ABB RobotStudio station: smART_ABB_robotstudio_model.rsstn

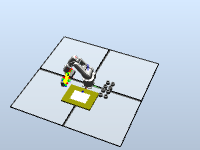
Station smART_v3 (saved by RobotStudio 6.7.7850.130)
Controller IRB120_3kg_0.58m
  mechanical unit ROB_1: IRB120_3_58__01, 6 joints, base frame (0, 0, 0) mm
Layout (positions relative to the parent item):
  - IRB120_3_58__01 [mechanism, from Robots\IRB120_3_58_G_01.rslib] at (0, 0, 0) mm; joint values [-1.4746, 0.7594, 0.252, 0.0074, 0.5575, -0.7708] (rad or m)
  - Grundplatte [part] at (-350, 0, 0) mm
  - Malplatte [part]
  - Papier [part]
  - Waschstation [part]
  - pen [mechanism] at (39.23, -403.71, 195) mm, rotated rx 179.91 ry 0.23 rz 139.31 deg
      TCP Pinsel at (1020, 52.5, 190) mm
      links: Pinsel
  - Pinselstation [part] at (-170, -459.8, 0) mm
  - Farben [part] at (162, 305.7, 0) mm
  - Frame_1 [frame] at (0, 0, 190) mm
Attachment: pen is attached to IRB120_3_58__01 / Link6
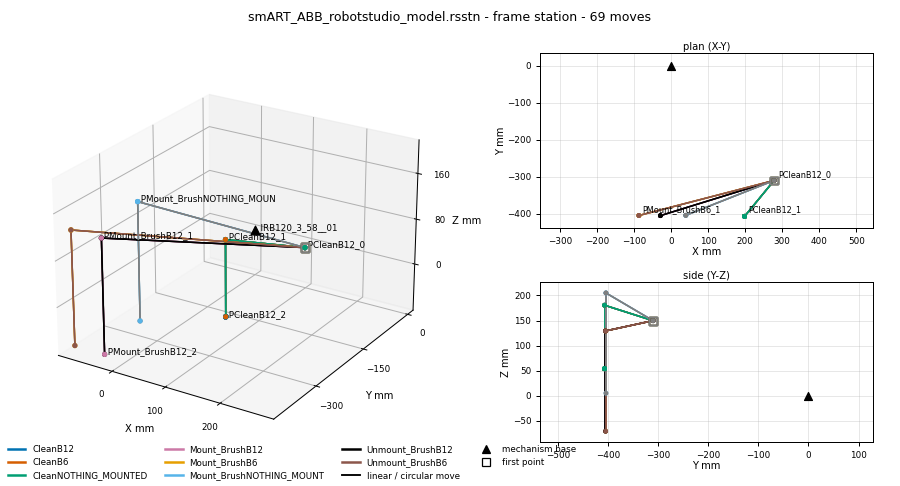
[picture p0: tool path of smART_ABB_robotstudio_model.rsstn in frame station, 69 of 69 moves have a stored position in this frame; points joined in program order, loops and branches not executed]
Targets, tools, work objects and paths stored in the station, written as RAPID:
! task T_ROB1
MODULE CalibData
  TASK PERS tooldata Tooldata_1:=[TRUE,[[0,0,0],[1,0,0,0]],[1,[0,0,1],[1,0,0,0],0,0,0]];
  PERS tooldata Pinsel:=[TRUE,[[0,0,190],[1,0,0,0]],[1,[0,0,1],[1,0,0,0],0,0,0]];
  TASK PERS wobjdata paintWO:=[FALSE,TRUE,"",[[242.9,0,0],[1,0,0,0]],[[0,0,0],[1,0,0,0]]];
  PERS tooldata pen:=[TRUE,[[0,0,190],[1,0,0,0]],[1,[0,0,1],[1,0,0,0],0,0,0]];
ENDMODULE

! task T_ROB1
MODULE Module1
  CONST robtarget PCleanB12_0:=[[35.2,-310,149.7],[0.00217,0.34764,0.93763,0],[0,0,0,0],[9E+09,9E+09,9E+09,9E+09,9E+09,9E+09]];
  CONST robtarget PCleanB12_1:=[[-44.4,-406.8,180.5],[0.00217,0.34764,0.93763,0],[0,0,0,0],[9E+09,9E+09,9E+09,9E+09,9E+09,9E+09]];
  CONST robtarget PCleanB12_2:=[[-44.4,-406.8,53.9],[0.00217,0.34764,0.93763,0],[0,0,0,0],[9E+09,9E+09,9E+09,9E+09,9E+09,9E+09]];
  CONST robtarget PCleanB12_3:=[[-44.4,-406.8,53.9],[0.00217,0.34764,0.93763,0],[0,0,0,0],[9E+09,9E+09,9E+09,9E+09,9E+09,9E+09]];
  CONST robtarget PCleanB12_4:=[[-44.4,-406.8,53.9],[0.00217,0.34764,0.93763,0],[0,0,0,0],[9E+09,9E+09,9E+09,9E+09,9E+09,9E+09]];
  CONST robtarget PCleanB6_0:=[[35.2,-310,149.7],[0.00217,0.34764,0.93763,0],[0,0,0,0],[9E+09,9E+09,9E+09,9E+09,9E+09,9E+09]];
  CONST robtarget PCleanB6_1:=[[-44.4,-406.8,180.5],[0.00217,0.34764,0.93763,0],[0,0,0,0],[9E+09,9E+09,9E+09,9E+09,9E+09,9E+09]];
  CONST robtarget PCleanB6_2:=[[-44.4,-406.8,53.9],[0.00217,0.34764,0.93763,0],[0,0,0,0],[9E+09,9E+09,9E+09,9E+09,9E+09,9E+09]];
  CONST robtarget PCleanB6_3:=[[-44.4,-406.8,53.9],[0.00217,0.34764,0.93763,0],[0,0,0,0],[9E+09,9E+09,9E+09,9E+09,9E+09,9E+09]];
  CONST robtarget PCleanB6_4:=[[-44.4,-406.8,53.9],[0.00217,0.34764,0.93763,0],[0,0,0,0],[9E+09,9E+09,9E+09,9E+09,9E+09,9E+09]];
  CONST robtarget PCleanNOTHING_MOUNTED_0:=[[35.2,-310,149.7],[0.00217,0.34764,0.93763,0],[0,0,0,0],[9E+09,9E+09,9E+09,9E+09,9E+09,9E+09]];
  CONST robtarget PCleanNOTHING_MOUNTED_1:=[[-44.4,-406.8,180.5],[0.00217,0.34764,0.93763,0],[0,0,0,0],[9E+09,9E+09,9E+09,9E+09,9E+09,9E+09]];
  CONST robtarget PCleanNOTHING_MOUNTED_2:=[[-44.4,-406.8,53.9],[0.00217,0.34764,0.93763,0],[0,0,0,0],[9E+09,9E+09,9E+09,9E+09,9E+09,9E+09]];
  CONST robtarget PCleanNOTHING_MOUNTED_3:=[[-44.4,-406.8,53.9],[0.00217,0.34764,0.93763,0],[0,0,0,0],[9E+09,9E+09,9E+09,9E+09,9E+09,9E+09]];
  CONST robtarget PCleanNOTHING_MOUNTED_4:=[[-44.4,-406.8,53.9],[0.00217,0.34764,0.93763,0],[0,0,0,0],[9E+09,9E+09,9E+09,9E+09,9E+09,9E+09]];
  CONST robtarget PMount_BrushB12_0:=[[35.2,-310,149.7],[0.00217,0.34764,0.93763,0],[0,0,0,0],[9E+09,9E+09,9E+09,9E+09,9E+09,9E+09]];
  CONST robtarget PMount_BrushB12_1:=[[-271.5,-404.9,129.2],[0.00217,0.34764,0.93763,0],[0,0,0,0],[9E+09,9E+09,9E+09,9E+09,9E+09,9E+09]];
  CONST robtarget PMount_BrushB12_2:=[[-271.5,-404.9,-70.8],[0.00217,0.34764,0.93763,0],[0,0,0,0],[9E+09,9E+09,9E+09,9E+09,9E+09,9E+09]];
  CONST robtarget PMount_BrushB12_3:=[[-271.5,-404.9,129.2],[0.00217,0.34764,0.93763,0],[0,0,0,0],[9E+09,9E+09,9E+09,9E+09,9E+09,9E+09]];
  CONST robtarget PMount_BrushB12_4:=[[35.2,-310,149.7],[0.00217,0.34764,0.93763,0],[0,0,0,0],[9E+09,9E+09,9E+09,9E+09,9E+09,9E+09]];
  CONST robtarget PMount_BrushB6_0:=[[35.2,-310,149.7],[0.00217,0.34764,0.93763,0],[0,0,0,0],[9E+09,9E+09,9E+09,9E+09,9E+09,9E+09]];
  CONST robtarget PMount_BrushB6_1:=[[-329.4,-404.5,129.2],[0.00217,0.34764,0.93763,0],[0,0,0,0],[9E+09,9E+09,9E+09,9E+09,9E+09,9E+09]];
  CONST robtarget PMount_BrushB6_2:=[[-329.4,-404.5,-70.8],[0.00217,0.34764,0.93763,0],[0,0,0,0],[9E+09,9E+09,9E+09,9E+09,9E+09,9E+09]];
  CONST robtarget PMount_BrushB6_3:=[[-329.4,-404.5,129.2],[0.00217,0.34764,0.93763,0],[0,0,0,0],[9E+09,9E+09,9E+09,9E+09,9E+09,9E+09]];
  CONST robtarget PMount_BrushB6_4:=[[35.2,-310,149.7],[0.00217,0.34764,0.93763,0],[0,0,0,0],[9E+09,9E+09,9E+09,9E+09,9E+09,9E+09]];
  CONST robtarget PMount_BrushNOTHING_MOUNTED_0:=[[35.2,-310,149.7],[0.00217,0.34764,0.93763,0],[0,0,0,0],[9E+09,9E+09,9E+09,9E+09,9E+09,9E+09]];
  CONST robtarget PMount_BrushNOTHING_MOUNTED_1:=[[-202.9,-404,205],[0.00217,0.34764,0.93763,0],[0,0,0,0],[9E+09,9E+09,9E+09,9E+09,9E+09,9E+09]];
  CONST robtarget PMount_BrushNOTHING_MOUNTED_2:=[[-202.9,-404,5],[0.00217,0.34764,0.93763,0],[0,0,0,0],[9E+09,9E+09,9E+09,9E+09,9E+09,9E+09]];
  CONST robtarget PMount_BrushNOTHING_MOUNTED_3:=[[-202.9,-404,205],[0.00217,0.34764,0.93763,0],[0,0,0,0],[9E+09,9E+09,9E+09,9E+09,9E+09,9E+09]];
  CONST robtarget PMount_BrushNOTHING_MOUNTED_4:=[[35.2,-310,149.7],[0.00217,0.34764,0.93763,0],[0,0,0,0],[9E+09,9E+09,9E+09,9E+09,9E+09,9E+09]];
  CONST robtarget PUnmount_BrushB12_0:=[[35.2,-310,149.7],[0.00217,0.34764,0.93763,0],[0,0,0,0],[9E+09,9E+09,9E+09,9E+09,9E+09,9E+09]];
  CONST robtarget PUnmount_BrushB12_1:=[[-271.5,-404.9,129.2],[0.00217,0.34764,0.93763,0],[0,0,0,0],[9E+09,9E+09,9E+09,9E+09,9E+09,9E+09]];
  CONST robtarget PUnmount_BrushB12_2:=[[-271.5,-404.9,-70.8],[0.00217,0.34764,0.93763,0],[0,0,0,0],[9E+09,9E+09,9E+09,9E+09,9E+09,9E+09]];
  CONST robtarget PUnmount_BrushB12_3:=[[-271.5,-404.9,129.2],[0.00217,0.34764,0.93763,0],[0,0,0,0],[9E+09,9E+09,9E+09,9E+09,9E+09,9E+09]];
  CONST robtarget PUnmount_BrushB12_4:=[[35.2,-310,149.7],[0.00217,0.34764,0.93763,0],[0,0,0,0],[9E+09,9E+09,9E+09,9E+09,9E+09,9E+09]];
  CONST robtarget PUnmount_BrushB6_0:=[[35.2,-310,149.7],[0.00217,0.34764,0.93763,0],[0,0,0,0],[9E+09,9E+09,9E+09,9E+09,9E+09,9E+09]];
  CONST robtarget PUnmount_BrushB6_1:=[[-329.4,-404.5,129.2],[0.00217,0.34764,0.93763,0],[0,0,0,0],[9E+09,9E+09,9E+09,9E+09,9E+09,9E+09]];
  CONST robtarget PUnmount_BrushB6_2:=[[-329.4,-404.5,-70.8],[0.00217,0.34764,0.93763,0],[0,0,0,0],[9E+09,9E+09,9E+09,9E+09,9E+09,9E+09]];
  CONST robtarget PUnmount_BrushB6_3:=[[-329.4,-404.5,129.2],[0.00217,0.34764,0.93763,0],[0,0,0,0],[9E+09,9E+09,9E+09,9E+09,9E+09,9E+09]];
  CONST robtarget PUnmount_BrushB6_4:=[[35.2,-310,149.7],[0.00217,0.34764,0.93763,0],[0,0,0,0],[9E+09,9E+09,9E+09,9E+09,9E+09,9E+09]];
  CONST robtarget PUnmount_BrushNOTHING_MOUNTED_0:=[[35.2,-310,149.7],[0.00217,0.34764,0.93763,0],[0,0,0,0],[9E+09,9E+09,9E+09,9E+09,9E+09,9E+09]];
  CONST robtarget PUnmount_BrushNOTHING_MOUNTED_1:=[[-202.9,-404,205],[0.00217,0.34764,0.93763,0],[0,0,0,0],[9E+09,9E+09,9E+09,9E+09,9E+09,9E+09]];
  CONST robtarget PUnmount_BrushNOTHING_MOUNTED_2:=[[-202.9,-404,5],[0.00217,0.34764,0.93763,0],[0,0,0,0],[9E+09,9E+09,9E+09,9E+09,9E+09,9E+09]];
  CONST robtarget PUnmount_BrushNOTHING_MOUNTED_3:=[[-202.9,-404,205],[0.00217,0.34764,0.93763,0],[0,0,0,0],[9E+09,9E+09,9E+09,9E+09,9E+09,9E+09]];
  CONST robtarget PCleanB12_5:=[[-44.4,-406.8,53.9],[0.00217,0.34764,0.93763,0],[0,0,0,0],[9E+09,9E+09,9E+09,9E+09,9E+09,9E+09]];
  CONST robtarget PCleanB12_6:=[[-44.4,-406.8,53.9],[0.00217,0.34764,0.93763,0],[0,0,0,0],[9E+09,9E+09,9E+09,9E+09,9E+09,9E+09]];
  CONST robtarget PCleanB12_7:=[[-44.4,-406.8,53.9],[0.00217,0.34764,0.93763,0],[0,0,0,0],[9E+09,9E+09,9E+09,9E+09,9E+09,9E+09]];
  CONST robtarget PCleanB12_8:=[[-44.4,-406.8,53.9],[0.00217,0.34764,0.93763,0],[0,0,0,0],[9E+09,9E+09,9E+09,9E+09,9E+09,9E+09]];
  CONST robtarget PCleanB12_11:=[[-44.4,-406.8,180.5],[0.00217,0.34764,0.93763,0],[0,0,0,0],[9E+09,9E+09,9E+09,9E+09,9E+09,9E+09]];
  CONST robtarget PCleanB12_12:=[[35.2,-310,149.7],[0.00217,0.34764,0.93763,0],[0,0,0,0],[9E+09,9E+09,9E+09,9E+09,9E+09,9E+09]];
  CONST robtarget PCleanB6_5:=[[-44.4,-406.8,53.9],[0.00217,0.34764,0.93763,0],[0,0,0,0],[9E+09,9E+09,9E+09,9E+09,9E+09,9E+09]];
  CONST robtarget PCleanB6_6:=[[-44.4,-406.8,53.9],[0.00217,0.34764,0.93763,0],[0,0,0,0],[9E+09,9E+09,9E+09,9E+09,9E+09,9E+09]];
  CONST robtarget PCleanB6_7:=[[-44.4,-406.8,53.9],[0.00217,0.34764,0.93763,0],[0,0,0,0],[9E+09,9E+09,9E+09,9E+09,9E+09,9E+09]];
  CONST robtarget PCleanB6_8:=[[-44.4,-406.8,53.9],[0.00217,0.34764,0.93763,0],[0,0,0,0],[9E+09,9E+09,9E+09,9E+09,9E+09,9E+09]];
  CONST robtarget PCleanB6_11:=[[-44.4,-406.8,180.5],[0.00217,0.34764,0.93763,0],[0,0,0,0],[9E+09,9E+09,9E+09,9E+09,9E+09,9E+09]];
  CONST robtarget PCleanB6_12:=[[35.2,-310,149.7],[0.00217,0.34764,0.93763,0],[0,0,0,0],[9E+09,9E+09,9E+09,9E+09,9E+09,9E+09]];
  CONST robtarget PCleanNOTHING_MOUNTED_5:=[[-44.4,-406.8,53.9],[0.00217,0.34764,0.93763,0],[0,0,0,0],[9E+09,9E+09,9E+09,9E+09,9E+09,9E+09]];
  CONST robtarget PCleanNOTHING_MOUNTED_6:=[[-44.4,-406.8,53.9],[0.00217,0.34764,0.93763,0],[0,0,0,0],[9E+09,9E+09,9E+09,9E+09,9E+09,9E+09]];
  CONST robtarget PCleanNOTHING_MOUNTED_7:=[[-44.4,-406.8,53.9],[0.00217,0.34764,0.93763,0],[0,0,0,0],[9E+09,9E+09,9E+09,9E+09,9E+09,9E+09]];
  CONST robtarget PCleanNOTHING_MOUNTED_8:=[[-44.4,-406.8,53.9],[0.00217,0.34764,0.93763,0],[0,0,0,0],[9E+09,9E+09,9E+09,9E+09,9E+09,9E+09]];
  CONST robtarget PCleanNOTHING_MOUNTED_11:=[[-44.4,-406.8,180.5],[0.00217,0.34764,0.93763,0],[0,0,0,0],[9E+09,9E+09,9E+09,9E+09,9E+09,9E+09]];
  CONST robtarget PCleanNOTHING_MOUNTED_12:=[[35.2,-310,149.7],[0.00217,0.34764,0.93763,0],[0,0,0,0],[9E+09,9E+09,9E+09,9E+09,9E+09,9E+09]];
  CONST robtarget PTowelB12_0:=[[-430.2,-173.7,71.3],[0.00217,0.34764,0.93763,0],[0,0,0,0],[9E+09,9E+09,9E+09,9E+09,9E+09,9E+09]];
  CONST robtarget PCleanB12_9:=[[-44.4,-406.8,53.9],[0.00217,0.34764,0.93763,0],[0,0,0,0],[9E+09,9E+09,9E+09,9E+09,9E+09,9E+09]];
  CONST robtarget PCleanB12_10:=[[-44.4,-406.8,53.9],[0.00217,0.34764,0.93763,0],[0,0,0,0],[9E+09,9E+09,9E+09,9E+09,9E+09,9E+09]];
  CONST robtarget PCleanB6_9:=[[-44.4,-406.8,53.9],[0.00217,0.34764,0.93763,0],[0,0,0,0],[9E+09,9E+09,9E+09,9E+09,9E+09,9E+09]];
  CONST robtarget PCleanB6_10:=[[-44.4,-406.8,53.9],[0.00217,0.34764,0.93763,0],[0,0,0,0],[9E+09,9E+09,9E+09,9E+09,9E+09,9E+09]];
  CONST robtarget PCleanNOTHING_MOUNTED_9:=[[-44.4,-406.8,53.9],[0.00217,0.34764,0.93763,0],[0,0,0,0],[9E+09,9E+09,9E+09,9E+09,9E+09,9E+09]];
  CONST robtarget PCleanNOTHING_MOUNTED_10:=[[-44.4,-406.8,53.9],[0.00217,0.34764,0.93763,0],[0,0,0,0],[9E+09,9E+09,9E+09,9E+09,9E+09,9E+09]];
  CONST robtarget PUnmount_BrushNOTHING_MOUNTED_4:=[[35.2,-310,149.7],[0.00217,0.34764,0.93763,0],[0,0,0,0],[9E+09,9E+09,9E+09,9E+09,9E+09,9E+09]];
  PROC main()
    SetDO do11,1;
    ChBrF_NOTHING_MOUNTED_TO_B12;
    CleanB12;
    CleanB12;
    CleanB12;
    CleanB12;
    CleanB12;
    CleanB12;
    ChBrF_B12_TO_B6;
    CleanB6;
    CleanB6;
    ChBrF_B6_TO_B12;
    CleanB12;
    CleanB12;
    CleanB12;
    CleanB12;
    ChBrF_B12_TO_B6;
    CleanB6;
    CleanB6;
    CleanB6;
    CleanB6;
    CleanB6;
    CleanB6;
    ChBrF_B6_TO_B12;
    CleanB12;
    CleanB12;
    CleanB12;
    CleanB12;
    ChBrF_B12_TO_B6;
    CleanB6;
    CleanB6;
    ChBrF_B6_TO_B12;
    CleanB12;
    CleanB12;
    CleanB12;
    CleanB12;
    CleanB12;
    CleanB12;
    ChBrF_B12_TO_B6;
    CleanB6;
    CleanB6;
    CleanB6;
    CleanB6;
    CleanB6;
    CleanB6;
    CleanB6;
    CleanB6;
    ChBrF_B6_TO_B12;
    CleanB12;
    CleanB12;
    ChBrF_B12_TO_B6;
    CleanB6;
    CleanB6;
    CleanB6;
    CleanB6;
    CleanB6;
    CleanB6;
    CleanB6;
    CleanB6;
    ChBrF_B6_TO_B12;
    CleanB12;
    CleanB12;
    CleanB12;
    CleanB12;
    CleanB12;
    CleanB12;
    CleanB12;
    CleanB12;
    CleanB12;
    CleanB12;
    ChBrF_B12_TO_B6;
    CleanB6;
    CleanB6;
    CleanB6;
    CleanB6;
    CleanB6;
    CleanB6;
    CleanB6;
    CleanB6;
    CleanB6;
    CleanB6;
    CleanB6;
    CleanB6;
    ChBrF_B6_TO_B12;
    CleanB12;
    CleanB12;
    CleanB12;
    CleanB12;
    CleanB12;
    CleanB12;
    CleanB12;
    CleanB12;
    CleanB12;
    CleanB12;
    ChBrF_B12_TO_B6;
    CleanB6;
    CleanB6;
    CleanB6;
    CleanB6;
    CleanB6;
    CleanB6;
    CleanB6;
    CleanB6;
    CleanB6;
    CleanB6;
    CleanB6;
    CleanB6;
    CleanB6;
    CleanB6;
    CleanB6;
    CleanB6;
    CleanB6;
    CleanB6;
    CleanB6;
    CleanB6;
    CleanB6;
    CleanB6;
    CleanB6;
    CleanB6;
    CleanB6;
    CleanB6;
    CleanB6;
    CleanB6;
    CleanB6;
    CleanB6;
    CleanB6;
    CleanB6;
    CleanB6;
    CleanB6;
    CleanB6;
    CleanB6;
    CleanB6;
    CleanB6;
    CleanB6;
    CleanB6;
    CleanB6;
    CleanB6;
    CleanB6;
    CleanB6;
    CleanB6;
    CleanB6;
    CleanB6;
    CleanB6;
    CleanB6;
    CleanB6;
    CleanB6;
    CleanB6;
    CleanB6;
    CleanB6;
    CleanB6;
    CleanB6;
    CleanB6;
    CleanB6;
    CleanB6;
    CleanB6;
    CleanB6;
    CleanB6;
    CleanB6;
    CleanB6;
    CleanB6;
    CleanB6;
    CleanB6;
    CleanB6;
    CleanB6;
    CleanB6;
    CleanB6;
    CleanB6;
    CleanB6;
    CleanB6;
    CleanB6;
    CleanB6;
    CleanB6;
    CleanB6;
    CleanB6;
    CleanB6;
    CleanB6;
    CleanB6;
    CleanB6;
    CleanB6;
    CleanB6;
    CleanB6;
    CleanB6;
    CleanB6;
    CleanB6;
    CleanB6;
    CleanB6;
    CleanB6;
    CleanB6;
    CleanB6;
    CleanB6;
    CleanB6;
    CleanB6;
    CleanB6;
    CleanB6;
    CleanB6;
    CleanB6;
    CleanB6;
    CleanB6;
    CleanB6;
    CleanB6;
    CleanB6;
    CleanB6;
    CleanB6;
    CleanB6;
    CleanB6;
    CleanB6;
    CleanB6;
    CleanB6;
    CleanB6;
    CleanB6;
    CleanB6;
    CleanB6;
    CleanB6;
    CleanB6;
    CleanB6;
    CleanB6;
    CleanB6;
    CleanB6;
    CleanB6;
    CleanB6;
    CleanB6;
    CleanB6;
    CleanB6;
    CleanB6;
    CleanB6;
    CleanB6;
    CleanB6;
    CleanB6;
    CleanB6;
    CleanB6;
    CleanB6;
    CleanB6;
    CleanB6;
    CleanB6;
    CleanB6;
    CleanB6;
    CleanB6;
    CleanB6;
    CleanB6;
    CleanB6;
    CleanB6;
    CleanB6;
    CleanB6;
    CleanB6;
    CleanB6;
    CleanB6;
    CleanB6;
    CleanB6;
    CleanB6;
    CleanB6;
    CleanB6;
    CleanB6;
    CleanB6;
    CleanB6;
    CleanB6;
    CleanB6;
    CleanB6;
    CleanB6;
    CleanB6;
    CleanB6;
    CleanB6;
    CleanB6;
    CleanB6;
    CleanB6;
    CleanB6;
    CleanB6;
    CleanB6;
    CleanB6;
    CleanB6;
    CleanB6;
    CleanB6;
    CleanB6;
    CleanB6;
    CleanB6;
    CleanB6;
    CleanB6;
    CleanB6;
    CleanB6;
    CleanB6;
    CleanB6;
    CleanB6;
    CleanB6;
    CleanB6;
    CleanB6;
    CleanB6;
    CleanB6;
    CleanB6;
    CleanB6;
    CleanB6;
    CleanB6;
    CleanB6;
    CleanB6;
    CleanB6;
    CleanB6;
    CleanB6;
    CleanB6;
    CleanB6;
    CleanB6;
    CleanB6;
    CleanB6;
    CleanB6;
    CleanB6;
    CleanB6;
    CleanB6;
    CleanB6;
    CleanB6;
    CleanB6;
    CleanB6;
    CleanB6;
    CleanB6;
    CleanB6;
    CleanB6;
    CleanB6;
    CleanB6;
    CleanB6;
    CleanB6;
    CleanB6;
    CleanB6;
    CleanB6;
    CleanB6;
    CleanB6;
    CleanB6;
    CleanB6;
    CleanB6;
    CleanB6;
    CleanB6;
    CleanB6;
    CleanB6;
    CleanB6;
    CleanB6;
    CleanB6;
    CleanB6;
    CleanB6;
    CleanB6;
    CleanB6;
    CleanB6;
    CleanB6;
    CleanB6;
    CleanB6;
    CleanB6;
    CleanB6;
    CleanB6;
    CleanB6;
    CleanB6;
    CleanB6;
    CleanB6;
    CleanB6;
    CleanB6;
    CleanB6;
    CleanB6;
    CleanB6;
    CleanB6;
    CleanB6;
    CleanB6;
    CleanB6;
    CleanB6;
    CleanB6;
    CleanB6;
    CleanB6;
    CleanB6;
    CleanB6;
    CleanB6;
    CleanB6;
    CleanB6;
    CleanB6;
    CleanB6;
    CleanB6;
    CleanB6;
    CleanB6;
    CleanB6;
    CleanB6;
    CleanB6;
    CleanB6;
    CleanB6;
    CleanB6;
    CleanB6;
    CleanB6;
    CleanB6;
    CleanB6;
    CleanB6;
    CleanB6;
    CleanB6;
    CleanB6;
    CleanB6;
    CleanB6;
    CleanB6;
    CleanB6;
    CleanB6;
    CleanB6;
    CleanB6;
    CleanB6;
    CleanB6;
    CleanB6;
    CleanB6;
    CleanB6;
    CleanB6;
    CleanB6;
    CleanB6;
    CleanB6;
    CleanB6;
    CleanB6;
    CleanB6;
    CleanB6;
    CleanB6;
    CleanB6;
    CleanB6;
    CleanB6;
    CleanB6;
    CleanB6;
    CleanB6;
    CleanB6;
    CleanB6;
    CleanB6;
    CleanB6;
    CleanB6;
    CleanB6;
    CleanB6;
    CleanB6;
    CleanB6;
    CleanB6;
    CleanB6;
    CleanB6;
    CleanB6;
    CleanB6;
    CleanB6;
    CleanB6;
    CleanB6;
    CleanB6;
    CleanB6;
    CleanB6;
    CleanB6;
    CleanB6;
    CleanB6;
    CleanB6;
    CleanB6;
    CleanB6;
    CleanB6;
    CleanB6;
    CleanB6;
    CleanB6;
    CleanB6;
    CleanB6;
    CleanB6;
    CleanB6;
    CleanB6;
    CleanB6;
    CleanB6;
    CleanB6;
    CleanB6;
    CleanB6;
    CleanB6;
    CleanB6;
    CleanB6;
    CleanB6;
    CleanB6;
    CleanB6;
    CleanB6;
    CleanB6;
    CleanB6;
    CleanB6;
    CleanB6;
    CleanB6;
    ChBrF_B6_TO_NOTHING_MOUNTED;
  ENDPROC
  PROC ChBrF_B12_TO_B6()
    Unmount_BrushB12;
    Mount_BrushB6;
  ENDPROC
  PROC ChBrF_B12_TO_NOTHING_MOUNTED()
    Unmount_BrushB12;
    Mount_BrushNOTHING_MOUNTED;
  ENDPROC
  PROC ChBrF_B6_TO_B12()
    Unmount_BrushB6;
    Mount_BrushB12;
  ENDPROC
  PROC ChBrF_B6_TO_NOTHING_MOUNTED()
    Unmount_BrushB6;
    Mount_BrushNOTHING_MOUNTED;
  ENDPROC
  PROC ChBrF_NOTHING_MOUNTED_TO_B12()
    Unmount_BrushNOTHING_MOUNTED;
    Mount_BrushB12;
  ENDPROC
  PROC ChBrF_NOTHING_MOUNTED_TO_B6()
    Unmount_BrushNOTHING_MOUNTED;
    Mount_BrushB6;
  ENDPROC
  PROC CleanB12()
    MoveL PCleanB12_0,v400,fine,pen\WObj:=paintWO;
    MoveL PCleanB12_1,v400,fine,pen\WObj:=paintWO;
    SetDO do10,1;
    SetDO do12,0;
    SetDO do13,0;
    SetDO do14,1;
    WaitTime 0.01;
    MoveL PCleanB12_2,v400,fine,pen\WObj:=paintWO;
    WaitTime 0.7777777777777778;
    MoveL PCleanB12_3,v300,fine,pen\WObj:=paintWO;
    WaitTime 0.7777777777777778;
    MoveL PCleanB12_4,v300,fine,pen\WObj:=paintWO;
    WaitTime 0.7777777777777778;
    MoveL PCleanB12_5,v300,fine,pen\WObj:=paintWO;
    WaitTime 0.7777777777777778;
    MoveL PCleanB12_6,v400,fine,pen\WObj:=paintWO;
    WaitTime 0.7777777777777778;
    MoveL PCleanB12_7,v300,fine,pen\WObj:=paintWO;
    WaitTime 0.7777777777777778;
    MoveL PCleanB12_8,v300,fine,pen\WObj:=paintWO;
    WaitTime 0.7777777777777778;
    MoveL PCleanB12_9,v300,fine,pen\WObj:=paintWO;
    WaitTime 0.7777777777777778;
    MoveL PCleanB12_10,v400,fine,pen\WObj:=paintWO;
    WaitTime 0.7777777777777778;
    SetDO do10,0;
    SetDO do12,0;
    SetDO do13,0;
    SetDO do14,0;
    MoveL PCleanB12_11,v400,fine,pen\WObj:=paintWO;
    MoveL PCleanB12_12,v400,fine,pen\WObj:=paintWO;
  ENDPROC
  PROC CleanB6()
    MoveL PCleanB6_0,v400,fine,pen\WObj:=paintWO;
    MoveL PCleanB6_1,v400,fine,pen\WObj:=paintWO;
    SetDO do10,1;
    SetDO do12,0;
    SetDO do13,0;
    SetDO do14,1;
    WaitTime 0.01;
    MoveL PCleanB6_2,v400,fine,pen\WObj:=paintWO;
    WaitTime 0.7777777777777778;
    MoveL PCleanB6_3,v300,fine,pen\WObj:=paintWO;
    WaitTime 0.7777777777777778;
    MoveL PCleanB6_4,v300,fine,pen\WObj:=paintWO;
    WaitTime 0.7777777777777778;
    MoveL PCleanB6_5,v300,fine,pen\WObj:=paintWO;
    WaitTime 0.7777777777777778;
    MoveL PCleanB6_6,v400,fine,pen\WObj:=paintWO;
    WaitTime 0.7777777777777778;
    MoveL PCleanB6_7,v300,fine,pen\WObj:=paintWO;
    WaitTime 0.7777777777777778;
    MoveL PCleanB6_8,v300,fine,pen\WObj:=paintWO;
    WaitTime 0.7777777777777778;
    MoveL PCleanB6_9,v300,fine,pen\WObj:=paintWO;
    WaitTime 0.7777777777777778;
    MoveL PCleanB6_10,v400,fine,pen\WObj:=paintWO;
    WaitTime 0.7777777777777778;
    SetDO do10,0;
    SetDO do12,0;
    SetDO do13,0;
    SetDO do14,0;
    MoveL PCleanB6_11,v400,fine,pen\WObj:=paintWO;
    MoveL PCleanB6_12,v400,fine,pen\WObj:=paintWO;
  ENDPROC
  PROC CleanNOTHING_MOUNTED()
    MoveL PCleanNOTHING_MOUNTED_0,v400,fine,pen\WObj:=paintWO;
    MoveL PCleanNOTHING_MOUNTED_1,v400,fine,pen\WObj:=paintWO;
    SetDO do10,1;
    SetDO do12,0;
    SetDO do13,0;
    SetDO do14,1;
    WaitTime 0.01;
    MoveL PCleanNOTHING_MOUNTED_2,v400,fine,pen\WObj:=paintWO;
    WaitTime 0.7777777777777778;
    MoveL PCleanNOTHING_MOUNTED_3,v300,fine,pen\WObj:=paintWO;
    WaitTime 0.7777777777777778;
    MoveL PCleanNOTHING_MOUNTED_4,v300,fine,pen\WObj:=paintWO;
    WaitTime 0.7777777777777778;
    MoveL PCleanNOTHING_MOUNTED_5,v300,fine,pen\WObj:=paintWO;
    WaitTime 0.7777777777777778;
    MoveL PCleanNOTHING_MOUNTED_6,v400,fine,pen\WObj:=paintWO;
    WaitTime 0.7777777777777778;
    MoveL PCleanNOTHING_MOUNTED_7,v300,fine,pen\WObj:=paintWO;
    WaitTime 0.7777777777777778;
    MoveL PCleanNOTHING_MOUNTED_8,v300,fine,pen\WObj:=paintWO;
    WaitTime 0.7777777777777778;
    MoveL PCleanNOTHING_MOUNTED_9,v300,fine,pen\WObj:=paintWO;
    WaitTime 0.7777777777777778;
    MoveL PCleanNOTHING_MOUNTED_10,v400,fine,pen\WObj:=paintWO;
    WaitTime 0.7777777777777778;
    SetDO do10,0;
    SetDO do12,0;
    SetDO do13,0;
    SetDO do14,0;
    MoveL PCleanNOTHING_MOUNTED_11,v400,fine,pen\WObj:=paintWO;
    MoveL PCleanNOTHING_MOUNTED_12,v400,fine,pen\WObj:=paintWO;
  ENDPROC
  PROC Mount_BrushB12()
    MoveL PMount_BrushB12_0,v400,fine,pen\WObj:=paintWO;
    MoveL PMount_BrushB12_1,v300,fine,pen\WObj:=paintWO;
    SetDO do4,1;
    MoveL PMount_BrushB12_2,v300,fine,pen\WObj:=paintWO;
    SetDO do4,0;
    WaitTime 0.8;
    MoveL PMount_BrushB12_3,v300,fine,pen\WObj:=paintWO;
    MoveL PMount_BrushB12_4,v400,fine,pen\WObj:=paintWO;
  ENDPROC
  PROC Mount_BrushB6()
    MoveL PMount_BrushB6_0,v400,fine,pen\WObj:=paintWO;
    MoveL PMount_BrushB6_1,v300,fine,pen\WObj:=paintWO;
    SetDO do4,1;
    MoveL PMount_BrushB6_2,v300,fine,pen\WObj:=paintWO;
    SetDO do4,0;
    WaitTime 0.8;
    MoveL PMount_BrushB6_3,v300,fine,pen\WObj:=paintWO;
    MoveL PMount_BrushB6_4,v400,fine,pen\WObj:=paintWO;
  ENDPROC
  PROC Mount_BrushNOTHING_MOUNTED()
    MoveL PMount_BrushNOTHING_MOUNTED_0,v400,fine,pen\WObj:=paintWO;
    MoveL PMount_BrushNOTHING_MOUNTED_1,v300,fine,pen\WObj:=paintWO;
    SetDO do4,1;
    MoveL PMount_BrushNOTHING_MOUNTED_2,v300,fine,pen\WObj:=paintWO;
    SetDO do4,0;
    WaitTime 0.8;
    MoveL PMount_BrushNOTHING_MOUNTED_3,v300,fine,pen\WObj:=paintWO;
    MoveL PMount_BrushNOTHING_MOUNTED_4,v400,fine,pen\WObj:=paintWO;
  ENDPROC
  PROC Unmount_BrushB12()
    MoveL PUnmount_BrushB12_0,v400,fine,pen\WObj:=paintWO;
    MoveL PUnmount_BrushB12_1,v300,fine,pen\WObj:=paintWO;
    MoveL PUnmount_BrushB12_2,v300,fine,pen\WObj:=paintWO;
    SetDO do4,1;
    WaitTime 0.8;
    MoveL PUnmount_BrushB12_3,v300,fine,pen\WObj:=paintWO;
    MoveL PUnmount_BrushB12_4,v400,fine,pen\WObj:=paintWO;
    SetDO do4,0;
  ENDPROC
  PROC Unmount_BrushB6()
    MoveL PUnmount_BrushB6_0,v400,fine,pen\WObj:=paintWO;
    MoveL PUnmount_BrushB6_1,v300,fine,pen\WObj:=paintWO;
    MoveL PUnmount_BrushB6_2,v300,fine,pen\WObj:=paintWO;
    SetDO do4,1;
    WaitTime 0.8;
    MoveL PUnmount_BrushB6_3,v300,fine,pen\WObj:=paintWO;
    MoveL PUnmount_BrushB6_4,v400,fine,pen\WObj:=paintWO;
    SetDO do4,0;
  ENDPROC
  PROC Unmount_BrushNOTHING_MOUNTED()
    MoveL PUnmount_BrushNOTHING_MOUNTED_0,v400,fine,pen\WObj:=paintWO;
    MoveL PUnmount_BrushNOTHING_MOUNTED_1,v300,fine,pen\WObj:=paintWO;
    MoveL PUnmount_BrushNOTHING_MOUNTED_2,v300,fine,pen\WObj:=paintWO;
    SetDO do4,1;
    WaitTime 0.8;
    MoveL PUnmount_BrushNOTHING_MOUNTED_3,v300,fine,pen\WObj:=paintWO;
    MoveL PUnmount_BrushNOTHING_MOUNTED_4,v400,fine,pen\WObj:=paintWO;
    SetDO do4,0;
  ENDPROC
ENDMODULE

